Omron CX-Programmer project NewProject (CX-Programmer 9.75)

# PLC NewPLC1: CP1L M

## Global symbols (name address type ; comment)
0.00 BOOL  ; Open
0.01 BOOL  ; Lock
0.02 BOOL  ; Emergency
0.03 BOOL  ; Overload
0.04 BOOL  ; Maju
0.05 BOOL  ; Mundur
0.06 BOOL  ; Kiri
0.07 BOOL  ; Kanan
0.08 BOOL  ; Naik
0.09 BOOL  ; Turun
100.00 BOOL  ; Hijau
100.01 BOOL  ; Merah
100.02 BOOL  ; M_Maju
100.03 BOOL  ; M_Mundur
100.04 BOOL  ; M_Kiri
100.05 BOOL  ; M_Kanan
100.06 BOOL  ; M_Naik
100.07 BOOL  ; M_Turun

## Program NewProgram1 (cyclic task 0)

### Section Section1

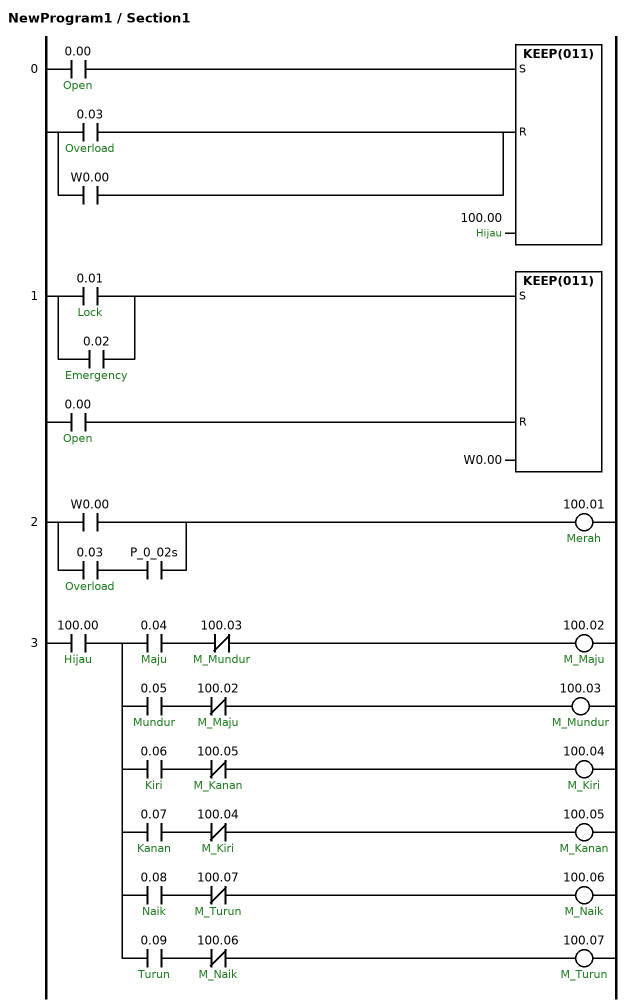
; rung 0
LD 0.00  ; Open
LD 0.03  ; Overload
OR W0.00
KEEP(011) 100.00  ; Hijau
; rung 1
LD 0.01  ; Lock
OR 0.02  ; Emergency
LD 0.00  ; Open
KEEP(011) W0.00
; rung 2
LD W0.00
LD 0.03  ; Overload
AND P_0_02s
ORLD
OUT 100.01  ; Merah
; rung 3
LD 100.00  ; Hijau
OUT TR0
AND 0.04  ; Maju
ANDNOT 100.03  ; M_Mundur
OUT 100.02  ; M_Maju
LD TR0
AND 0.05  ; Mundur
ANDNOT 100.02  ; M_Maju
OUT 100.03  ; M_Mundur
LD TR0
AND 0.06  ; Kiri
ANDNOT 100.05  ; M_Kanan
OUT 100.04  ; M_Kiri
LD TR0
AND 0.07  ; Kanan
ANDNOT 100.04  ; M_Kiri
OUT 100.05  ; M_Kanan
LD TR0
AND 0.08  ; Naik
ANDNOT 100.07  ; M_Turun
OUT 100.06  ; M_Naik
LD TR0
AND 0.09  ; Turun
ANDNOT 100.06  ; M_Naik
OUT 100.07  ; M_Turun

### Section END
; rung 0
END(001)